TYPE U_AXIS_GEAR_IN :
UNION

  stCtrl              : ARRAY[1..MAX_AXIS] OF ST_GEAR_IN;

  byCtrl    AT %I*    : ARRAY[1..MAX_AXIS] OF
                        ARRAY[1..SIZEOF(ST_GEAR_IN)] OF BYTE;
END_UNION
END_TYPE

(* stored: Version 1.1.0.1, ProductVersion 3.1.4026.13
   DUT U_AXIS_GEAR_IN: Id {b7da2e13-202f-0e79-190e-3874455a40fc} *)
